{attribute 'qualified_only'}
VAR_GLOBAL
	bProjectB : BOOL;
END_VAR

(* stored: Version 1.1.0.1, ProductVersion 3.1.4022.18
   GVL GVL_ProjectB: Id {b116bff9-cd44-4e40-b1dd-f859c1230760} *)
